(* CODESYS project semaforo.project

Project tree, tasks and I/O mapping:
  Device : CODESYS Control Win V3, 3S - Smart Software Solutions GmbH, order no. 305021, version 3.5.11.30
    application Application
      libraries: Standard, * (System)
      task MainTask (cyclic, interval t#20ms, priority 1) calls PLC_PRG
      program PLC_PRG [ST]
*)

// Device/Application/PLC_PRG
PROGRAM PLC_PRG
VAR
	start : BOOL;
	aux1 : BOOL;
	
	s1verde : BOOL;
	s1amarelo: BOOL;
	s1vermelho: BOOL; 
	
	s2verde : BOOL;
	s2amarelo: BOOL;
	s2vermelho: BOOL; 
	
	s3verde : BOOL;
	s3amarelo: BOOL;
	s3vermelho: BOOL; 
	
	s4azul: BOOL;
	
	t1: TOF;
	t2: TOF;
	t3: TOF;
	t4: TOF;
	t5: TOF;
	tstopOn: TP;
	tstopOf: TOF;
	
	time1: TIME;
	time2: TIME;
	time3: TIME;
	time4: TIME;
	time5: TIME;
	time6: TIME;
	time7: TIME;
	
	q1: BOOL;
	q2: BOOL;
	q3: BOOL;
	q4: BOOL;
	q5: BOOL;
	q6: BOOL;
	q7: BOOL;
	
	RSTART: R_TRIG;
	R1: R_TRIG;
	R3: R_TRIG;
	R4: R_TRIG;
	R5: R_TRIG;
	R6: R_TRIG;
	R7: R_TRIG;
	R8: R_TRIG;
END_VAR

IF start THEN 
	aux1 := TRUE;
ELSE
	aux1 := FALSE;
	s4azul:=FALSE;
		
	s1vermelho:=FALSE;
	s1verde:=FALSE;
	
	s2verde:=FALSE;
	s2vermelho:= FALSE;
	
	s3vermelho:=FALSE;
	s3verde:=FALSE;
	
	tstopOn(IN:= R6.Q OR R7.Q, PT:=T#1S,ET=>time6, Q=>q6);
	tstopOf(IN:= R8.Q, PT:=T#1S,ET=>time7, Q=>q7);
	IF Q6 THEN
		s1amarelo:=TRUE;
		s2amarelo:=TRUE;
		s3amarelo:=TRUE;
	END_IF
	
	
	IF Q7 THEN
		s1amarelo:=FALSE;
		s2amarelo:=FALSE;
		s3amarelo:=FALSE;
	END_IF
END_IF

IF aux1 THEN 
	t1(IN:=RSTART.Q OR R5.Q, PT:=T#15S,ET=>time1, Q=>q1);
	t2(IN:=R1.Q, PT:=T#15S,ET=>time2, Q=>q2);
	t3(IN:=R1.Q, PT:=T#5S,ET=>time3, Q=>q3);
	t4(IN:=R3.Q, PT:=T#10S,ET=>time4, Q=>q4);
	t5(IN:=r4.Q, PT:=T#5S,ET=>time5, Q=>q5);
	s1amarelo:=FALSE;
	s2amarelo:=FALSE;
	s3amarelo:=FALSE;
	IF q1 THEN 
		s1verde:=TRUE;	
		s1amarelo:=FALSE;	
		s1vermelho:=FALSE;
		
		s2vermelho:=TRUE;
		s2verde:=FALSE;
		s2amarelo:=FALSE;
		
		s3vermelho:=TRUE;	
		s3verde:=FALSE;	
		s3amarelo:=FALSE;	
	END_IF
		
	IF q2 THEN 
		s1verde:=FALSE;		
		s2vermelho:=FALSE;
		s2verde:=TRUE;
		s2amarelo:=FALSE;
		s3vermelho:=FALSE;	
		s3verde:=TRUE;	
		s3amarelo:=FALSE;
	END_IF
	
	IF q3 THEN 
		s1amarelo:=TRUE;
	END_IF
	
	if q4 then 
		s1vermelho:=true;
		s1amarelo:=false;
	END_IF
	
	IF q5 THEN 
		s4azul:=TRUE;
		
		s1vermelho:=TRUE;
		s1amarelo:=FALSE;
		s1verde:=FALSE;
		
		s2verde:=TRUE;
		s2vermelho:= FALSE;
		s2amarelo:=FALSE;
		
		s3vermelho:=TRUE;
		s3verde:=FALSE;
		s3amarelo:=FALSE;
	END_IF
END_IF
RSTART(CLK:=START);
R1(CLK:=NOT(Q1));
R3(CLK:=NOT(Q3));
R4(CLK:=NOT(Q4));
R5(CLK:=NOT(Q5));
R6(CLK :=NOT(START));
R7(CLK :=NOT(Q7));
R8(CLK :=NOT(Q6));

END_PROGRAM
